(* CoDeSys 2.3.9.31 project: 1floor_2014_05_04.pr6 *)
(* Libraries: TcPlcUtilitiesBC.lb6 13.5.05 12:19:40, PlcSystemBC.lb6 21.3.01 12:03:02, TcAdsBC.lb6 5.7.02 12:03:02, standard.lb6 5.6.98 12:03:02 *)

(* Global variable list: main *)
VAR_GLOBAL


(*ADS*)

	ads_adr1: STRING:='10.0.5.61.1.1';
	ads_adr2: STRING:='10.0.5.62.1.1';
	ads_adr3: STRING:='10.0.5.63.1.1';

	write_ads: ADSWRITE;

	data2floor: ARRAY[0..3] OF BYTE;
	data2floor_prev :ARRAY[0..3] OF BYTE;
	data3floor: ARRAY[0..10] OF BYTE;
	data3floor_prev :ARRAY[0..10] OF BYTE;

	m_fancoil_vitalnya_low 	AT%MX300.0: BOOL;
	m_fancoil_vitalnya_med 	AT%MX300.1: BOOL;
	m_fancoil_vitalnya_high 	AT%MX300.2: BOOL;
	skvazhyna 		AT%MX300.3:BOOL;
	tepla_pidloga		AT%MX300.4:BOOL;
	T_out3			AT%MB303:BYTE;


	iHour			AT%MB304:BYTE;
	iMinute			AT%MB305:BYTE;
	lights			AT%MB306:DWORD;

	sw_tambur2_1	AT%MX200.0:BOOL;
	sw_tambur3_2	AT%MX300.1:BOOL;
	bDarkOutside		AT%MX300.6:BOOL;
	bT_out_sign		AT%MX300.7:BOOL;

	eib_komora_l 						AT%MX400.0:BOOL;
	eib_su1_l 							AT%MX400.1:BOOL;
	eib_topochna_l 						AT%MX400.2:BOOL;
	eib_su2_bra	 						AT%MX400.3:BOOL;
	eib_topochna2_l 						AT%MX400.4:BOOL;
	eib_su2_l 							AT%MX400.5:BOOL;
	eib_su1_rakovyna 					AT%MX400.6:BOOL;
	eib_su2_dush 						AT%MX400.7:BOOL;
	eib_dush 							AT%MX401.0:BOOL;
	eib_vitalnya_smugy2 					AT%MX401.1:BOOL;
	eib_su2_polytsi 						AT%MX401.2:BOOL;
	eib_kuhnya1	 						AT%MX401.3:BOOL;
	eib_kuhnya2	 						AT%MX401.4:BOOL;
	eib_vitalnya_smugy1 					AT%MX401.5:BOOL;
	eib_vitalnya_l 						AT%MX401.6:BOOL;
	eib_vitalnya_prokladka 				AT%MX401.7:BOOL;
	eib_terassa_stina	 					AT%MX402.0:BOOL;
	eib_pidval_shody	 					AT%MX402.1:BOOL;
	eib_terassa 							AT%MX402.2:BOOL;
	eib_skhody2pov 						AT%MX402.3:BOOL;
	eib_tambur_l 							AT%MX402.4:BOOL;

	eib_vent_su1 							AT%MX402.5:BOOL;
	eib_vent_kuh_low 						AT%MX402.6:BOOL;
	eib_vent_dush 						AT%MX402.7:BOOL;
	eib_vent_komora 						AT%MX403.0:BOOL;
	eib_vent_kuh_high 					AT%MX403.1:BOOL;

END_VAR

(* Global variable list: physical *)
VAR_GLOBAL
(*din1_1*)moove_su1		AT %IX80.0:	BOOL;
(*din1_2*)moove_topochna	AT %IX80.1:	BOOL;
(*din1_3*)moove_su2	AT %IX80.2:	BOOL;
(*din1_4*)moove_korydor_ops	AT %IX80.3:	BOOL;
(*din1_5*)moove_korydor	AT %IX80.4:	BOOL;
(*din1_6*)moove_vitalnya	AT %IX80.5:	BOOL;
(*din1_7*)moove_komora	AT %IX80.6:	BOOL;
	din1_8	AT %IX80.7:	BOOL;
(*din2_1*)moove_kino		AT %IX81.0:	BOOL;
(*din2_2*)moove_skhody2_3	AT %IX81.1:	BOOL;
(*din2_3*)moove_skhody1_2	AT %IX81.2:	BOOL;
(*din2_4*)moove_garderob	AT %IX81.3:	BOOL;
(*din2_5*)moove_studio		AT %IX81.4:	BOOL;
(*din2_6*)moove_tambur3	AT %IX81.5:	BOOL;
(*din2_7*)moove_kabinet	AT %IX81.6:	BOOL;
(*din2_8*)moove_dytjacha	AT %IX81.7:	BOOL;
(*din3_1*)moove_spalnya	AT %IX82.0:	BOOL;
	din3_2	AT %IX82.1:	BOOL;
(*din3_3*)moove_korydor3	AT %IX82.2:	BOOL;
	din3_4	AT %IX82.3:	BOOL;
	din3_5	AT %IX82.4:	BOOL;
	din3_6	AT %IX82.5:	BOOL;
	din3_7	AT %IX82.6:	BOOL;
	(*din3_8sw_vhid2		AT %IX82.7:	BOOL;*)
	din4_1	AT %IX83.0:	BOOL;
	(*din4_2*)sw_su1_2		AT %IX83.1:	BOOL;
	(*din4_3*)sw_komora1		AT %IX83.2:	BOOL;
	(*din4_4*)sw_vhid1		AT %IX83.3:	BOOL;
	(*din4_5*)sw_topochna2	AT %IX83.4:	BOOL;
	sw_vhid2					AT %IX83.5:	BOOL;
	(*din4_7*)sw_topochna1	AT %IX83.6:	BOOL;
	(*din4_8*)sw_su1_1		AT %IX83.7:	BOOL;
	(*din5_1*)sw_tambur1_2	AT %IX84.0:	BOOL;
	(*din5_2*)sw_su2			AT %IX84.1:	BOOL;
	(*din5_3*)sw_kuh_su2		AT %IX84.2:	BOOL;
	(*din5_4*)sw_kuh3			AT %IX84.3:	BOOL;
	din5_5					AT %IX84.4:	BOOL;
	(*din5_6*)sw_kuh4			AT %IX84.5:	BOOL;
	(*din5_7*)sw_tambur1		AT %IX84.6:	BOOL;
	(*din5_8*)sw_vitalnya1		AT %IX84.7:	BOOL;
	(*din6_1*)sw_vitalnya2		AT %IX85.0:	BOOL;
	(*din6_2*)sw_kuh2			AT %IX85.1:	BOOL;
	din6_3					AT %IX85.2:	BOOL;
	(*din6_4*)sw_kuh1			AT %IX85.3:	BOOL;
	(*din6_5*)sw_vitalnya3		AT %IX85.4:	BOOL;
	(*din6_6*)sw_tambur3		AT %IX85.5:	BOOL;
	(*din6_7*)sw_tambur_su	AT %IX85.6:	BOOL;
	(*din6_8*)sw_transit2pov	AT %IX85.7:	BOOL;

(*din7_1*)ch_sensor1	AT %IX86.0:	BOOL;
(*din7_2*)ch_sensor2	AT %IX86.1:	BOOL;
(*din7_3*)zatoplennya_kot	AT %IX86.2:	BOOL;
(*din7_4*)zatoplennya_komora	AT %IX86.3:	BOOL;
(*din7_5*)zatoplennya_su2	AT %IX86.4:	BOOL;
(*din7_6*)zatoplennya_kuh	AT %IX86.5:	BOOL;
(*din7_7*)zatoplennya_su3pov	AT %IX86.6:	BOOL;
	din7_8	AT %IX86.7:	BOOL;

	(*dout1_1*)komora_l			AT %QX80.0:	BOOL;
	(*dout1_2*)su1_l				AT %QX80.1:	BOOL;
	(*dout1_3*)topochna_l			AT %QX80.2:	BOOL;
	(*dout1_4*)su2_bra			AT %QX80.3:	BOOL;
	(*dout1_5*)topochna2_l			AT %QX80.4:	BOOL;
	(*dout1_6*)su2_l				AT %QX80.5:	BOOL;
	(*dout1_7*)su1_rakovyna		AT %QX80.6:	BOOL;
	(*dout1_8*)su2_dush			AT %QX80.7:	BOOL;
	(*dout2_1*)dush				AT %QX81.0:	BOOL;
	(*dout2_2*)vitalnya_smugy2		AT %QX81.1:	BOOL;
	(*dout2_3*) su2_polytsi			AT %QX81.2:	BOOL;
	(*dout2_4*)fancoil_vitalnya_low			AT %QX81.3:	BOOL;
	(*dout2_5*)kuhnya1			AT %QX81.4:	BOOL;
	(*dout2_6*)fancoil_vitalnya_med			AT %QX81.5:	BOOL;
	(*dout2_7*)kuhnya2			AT %QX81.6:	BOOL;
	(*dout2_8*)fancoil_vitalnya_high		AT %QX81.7:	BOOL;
	w_valve_recirc	AT %QX82.0:	BOOL;
	dout3_2	AT %QX82.1:	BOOL;
	w_valve3pov	AT %QX82.2:	BOOL;
	(*dout3_4*)vitalnya_smugy1		AT %QX82.3:	BOOL;
	w_valve1pov	AT %QX82.4:	BOOL;
	(*dout3_6*)vitalnya_l			AT %QX82.5:	BOOL;
	(*dout3_7*)freecooling	AT %QX82.6:	BOOL;
	(*dout3_8*)vitalnya_prokladka	AT %QX82.7:	BOOL;
	(*dout4_1*)terassa_stina		AT %QX83.0:	BOOL;
	(*dout4_2*)pidval_shody		AT %QX83.1:	BOOL;
	(*dout4_3*)terassa				AT %QX83.2:	BOOL;
	(*dout4_4*)skhody2pov			AT %QX83.3:	BOOL;
	dout4_5	AT %QX83.4:	BOOL;
	dout4_6	AT %QX83.5:	BOOL;
	dout4_7	AT %QX83.6:	BOOL;
	(*dout4_8*)tambur_l			AT %QX83.7:	BOOL;
	dout5_1	AT %QX84.0:	BOOL;
	dout5_2 AT %QX84.1:	BOOL;
(*dout5_3*)gas_valve	AT %QX84.2:	BOOL;
	dout5_4	AT %QX84.3:	BOOL;
	dout5_5	AT %QX84.4:	BOOL;
	dout5_6	AT %QX84.5:	BOOL;
	dout5_7	AT %QX84.6:	BOOL;
	dout5_8	AT %QX84.7:	BOOL;
	dout6_1	AT %QX85.0:	BOOL;
	dout6_2	AT %QX85.1:	BOOL;
	dout6_3	AT %QX85.2:	BOOL;
	dout6_4	AT %QX85.3:	BOOL;
	dout6_5	AT %QX85.4:	BOOL;
	dout6_6	AT %QX85.5:	BOOL;
	dout6_7	AT %QX85.6:	BOOL;
	dout6_8	AT %QX85.7:	BOOL;
	dout7_1	AT %QX86.0:	BOOL;
	dout7_2	AT %QX86.1:	BOOL;
	dout7_3	AT %QX86.2:	BOOL;
	dout7_4	AT %QX86.3:	BOOL;
	dout7_5	AT %QX86.4:	BOOL;
	dout7_6	AT %QX86.5:	BOOL;
	dout7_7	AT %QX86.6:	BOOL;
	dout7_8	AT %QX86.7:	BOOL;
	dout8_1	AT %QX87.0:	BOOL;
	dout8_2	AT %QX87.1:	BOOL;
	dout8_3	AT %QX87.2:	BOOL;
	dout8_4	AT %QX87.3:	BOOL;
	dout8_5	AT %QX87.4:	BOOL;
	dout8_6	AT %QX87.5:	BOOL;
	dout8_7	AT %QX87.6:	BOOL;
	dout8_8	AT %QX87.7:	BOOL;
	(*dout9_1*)vent_su1		AT %QX88.0:	BOOL;
	(*dout9_2*)vent_kuh_low	AT %QX88.1:	BOOL;
	(*dout9_3*)vent_dush		AT %QX88.2:	BOOL;
	(*dout9_4*)collector_komora		AT %QX88.3:	BOOL;
	(*dout9_5*)vent_komora	AT %QX88.4:	BOOL;
	(*dout9_6	*)collector_kuh		AT %QX88.5:	BOOL;
	(*dout9_7*)vent_kuh_high	AT %QX88.6:	BOOL;
	(*dout9_8*)collector_vitalnya1	AT %QX88.7:	BOOL;
	(*dout10_1*)collector_vitalnya2	AT %QX89.0:	BOOL;
	dout10_2	AT %QX89.1:	BOOL;
	(*dout10_3*)collector_su2		AT %QX89.2:	BOOL;
	dout10_4	AT %QX89.3:	BOOL;
	(*dout10_5*)collector_vhid_stina	AT %QX89.4:	BOOL;
	dout10_6	AT %QX89.5:	BOOL;
	(*dout10_7*)collector_vhid		AT %QX89.6:	BOOL;
	dout10_8	AT %QX89.7:	BOOL;
	dout11_1	AT %QX90.0:	BOOL;
	dout11_2	AT %QX90.1:	BOOL;
	dout11_3	AT %QX90.2:	BOOL;
	dout11_4	AT %QX90.3:	BOOL;
	dout11_5	AT %QX90.4:	BOOL;
	dout11_6	AT %QX90.5:	BOOL;
	dout11_7	AT %QX90.6:	BOOL;
	dout11_8	AT %QX90.7:	BOOL;

	klapan_vitalnya	AT %QB2:	INT;
	KL4414_2_Out	AT %QB6:	INT;
	KL4414_3_Out	AT %QB10:	INT;
	KL4414_4_Out	AT %QB14:	INT;

	temp_vhid	AT %IB50:	INT; (*25*)
	temp_dush	AT %IB58:	INT;(*25*)
	temp_kuh	AT %IB66:	INT;(*-136*)
	temp_vhid_stina	AT %IB70:	INT;(*0*)
(*
(* @GLOBAL_VARIABLE_LIST := TwinCAT_Import *)
(* @PATH := '' *)
VAR_GLOBAL (* DO NOT CHANGE THIS SHEET MANUALLY! *)
	PlcInVar_0	AT %QB128:	USINT;
	PlcInVar_1	AT %QB129:	USINT;
	PlcInVar_2	AT %QB130:	USINT;
	PlcInVar_3	AT %QB131:	USINT;
	PlcInVar_4	AT %QB132:	USINT;
	PlcInVar_5	AT %QB133:	USINT;
	PlcInVar_6	AT %QB134:	USINT;
	PlcInVar_7	AT %QB135:	USINT;
	PlcInVar_8	AT %QB136:	USINT;
	PlcInVar_9	AT %QB137:	USINT;
	PlcInVar_10	AT %QB138:	USINT;
	PlcInVar_11	AT %QB139:	USINT;
	PlcInVar_12	AT %QB140:	USINT;
	PlcInVar_13	AT %QB141:	USINT;
	PlcInVar_14	AT %QB142:	USINT;
	PlcInVar_15	AT %QB143:	USINT;
	PlcOutVar_0	AT %IB128:	USINT;
	PlcOutVar_1	AT %IB129:	USINT;
	PlcOutVar_2	AT %IB130:	USINT;
	PlcOutVar_3	AT %IB131:	USINT;
	PlcOutVar_4	AT %IB132:	USINT;
	PlcOutVar_5	AT %IB133:	USINT;
	PlcOutVar_6	AT %IB134:	USINT;
	PlcOutVar_7	AT %IB135:	USINT;
	PlcOutVar_8	AT %IB136:	USINT;
	PlcOutVar_9	AT %IB137:	USINT;
	PlcOutVar_10	AT %IB138:	USINT;
	PlcOutVar_11	AT %IB139:	USINT;
	PlcOutVar_12	AT %IB140:	USINT;
	PlcOutVar_13	AT %IB141:	USINT;
	PlcOutVar_14	AT %IB142:	USINT;
	PlcOutVar_15	AT %IB143:	USINT;
	Term_2_KL4414_1_State	AT %IB0:	USINT;
	Term_2_KL4414_1_Data_In	AT %IB2:	INT;
	Term_2_KL4414_1_Ctrl	AT %QB0:	USINT;
	Term_2_KL4414_1_Data_Out	AT %QB2:	INT;
	Term_2_KL4414_2_State	AT %IB4:	USINT;
	Term_2_KL4414_2_Data_In	AT %IB6:	INT;
	Term_2_KL4414_2_Ctrl	AT %QB4:	USINT;
	Term_2_KL4414_2_Data_Out	AT %QB6:	INT;
	Term_2_KL4414_3_State	AT %IB8:	USINT;
	Term_2_KL4414_3_Data_In	AT %IB10:	INT;
	Term_2_KL4414_3_Ctrl	AT %QB8:	USINT;
	Term_2_KL4414_3_Data_Out	AT %QB10:	INT;
	Term_2_KL4414_4_State	AT %IB12:	USINT;
	Term_2_KL4414_4_Data_In	AT %IB14:	INT;
	Term_2_KL4414_4_Ctrl	AT %QB12:	USINT;
	Term_2_KL4414_4_Data_Out	AT %QB14:	INT;
	Term_14_KL3228_4_1_State	AT %IB16:	USINT;
	Term_14_KL3228_4_1_Data_In	AT %IB18:	INT;
	Term_14_KL3228_4_1_Ctrl	AT %QB16:	USINT;
	Term_14_KL3228_4_1_Data_Out	AT %QB18:	INT;
	Term_14_KL3228_4_2_State	AT %IB20:	USINT;
	Term_14_KL3228_4_2_Data_In	AT %IB22:	INT;
	Term_14_KL3228_4_2_Ctrl	AT %QB20:	USINT;
	Term_14_KL3228_4_2_Data_Out	AT %QB22:	INT;
	Term_14_KL3228_4_3_State	AT %IB24:	USINT;
	Term_14_KL3228_4_3_Data_In	AT %IB26:	INT;
	Term_14_KL3228_4_3_Ctrl	AT %QB24:	USINT;
	Term_14_KL3228_4_3_Data_Out	AT %QB26:	INT;
	Term_14_KL3228_4_4_State	AT %IB28:	USINT;
	Term_14_KL3228_4_4_Data_In	AT %IB30:	INT;
	Term_14_KL3228_4_4_Ctrl	AT %QB28:	USINT;
	Term_14_KL3228_4_4_Data_Out	AT %QB30:	INT;
	Term_15_KL3228_4_1_State	AT %IB32:	USINT;
	Term_15_KL3228_4_1_Data_In	AT %IB34:	INT;
	Term_15_KL3228_4_1_Ctrl	AT %QB32:	USINT;
	Term_15_KL3228_4_1_Data_Out	AT %QB34:	INT;
	Term_15_KL3228_4_2_State	AT %IB36:	USINT;
	Term_15_KL3228_4_2_Data_In	AT %IB38:	INT;
	Term_15_KL3228_4_2_Ctrl	AT %QB36:	USINT;
	Term_15_KL3228_4_2_Data_Out	AT %QB38:	INT;
	Term_15_KL3228_4_3_State	AT %IB40:	USINT;
	Term_15_KL3228_4_3_Data_In	AT %IB42:	INT;
	Term_15_KL3228_4_3_Ctrl	AT %QB40:	USINT;
	Term_15_KL3228_4_3_Data_Out	AT %QB42:	INT;
	Term_15_KL3228_4_4_State	AT %IB44:	USINT;
	Term_15_KL3228_4_4_Data_In	AT %IB46:	INT;
	Term_15_KL3228_4_4_Ctrl	AT %QB44:	USINT;
	Term_15_KL3228_4_4_Data_Out	AT %QB46:	INT;
	Term_16_KL3228_4_1_State	AT %IB48:	USINT;
	Term_16_KL3228_4_1_Data_In	AT %IB50:	INT;
	Term_16_KL3228_4_1_Ctrl	AT %QB48:	USINT;
	Term_16_KL3228_4_1_Data_Out	AT %QB50:	INT;
	Term_16_KL3228_4_2_State	AT %IB52:	USINT;
	Term_16_KL3228_4_2_Data_In	AT %IB54:	INT;
	Term_16_KL3228_4_2_Ctrl	AT %QB52:	USINT;
	Term_16_KL3228_4_2_Data_Out	AT %QB54:	INT;
	Term_16_KL3228_4_3_State	AT %IB56:	USINT;
	Term_16_KL3228_4_3_Data_In	AT %IB58:	INT;
	Term_16_KL3228_4_3_Ctrl	AT %QB56:	USINT;
	Term_16_KL3228_4_3_Data_Out	AT %QB58:	INT;
	Term_16_KL3228_4_4_State	AT %IB60:	USINT;
	Term_16_KL3228_4_4_Data_In	AT %IB62:	INT;
	Term_16_KL3228_4_4_Ctrl	AT %QB60:	USINT;
	Term_16_KL3228_4_4_Data_Out	AT %QB62:	INT;
	Term_17_KL3228_4_1_State	AT %IB64:	USINT;
	Term_17_KL3228_4_1_Data_In	AT %IB66:	INT;
	Term_17_KL3228_4_1_Ctrl	AT %QB64:	USINT;
	Term_17_KL3228_4_1_Data_Out	AT %QB66:	INT;
	Term_17_KL3228_4_2_State	AT %IB68:	USINT;
	Term_17_KL3228_4_2_Data_In	AT %IB70:	INT;
	Term_17_KL3228_4_2_Ctrl	AT %QB68:	USINT;
	Term_17_KL3228_4_2_Data_Out	AT %QB70:	INT;
	Term_17_KL3228_4_3_State	AT %IB72:	USINT;
	Term_17_KL3228_4_3_Data_In	AT %IB74:	INT;
	Term_17_KL3228_4_3_Ctrl	AT %QB72:	USINT;
	Term_17_KL3228_4_3_Data_Out	AT %QB74:	INT;
	Term_17_KL3228_4_4_State	AT %IB76:	USINT;
	Term_17_KL3228_4_4_Data_In	AT %IB78:	INT;
	Term_17_KL3228_4_4_Ctrl	AT %QB76:	USINT;
	Term_17_KL3228_4_4_Data_Out	AT %QB78:	INT; 
	Term_3_KL2408_1_Output	AT %QX80.0:	BOOL;
	Term_3_KL2408_2_Output	AT %QX80.1:	BOOL;
	Term_3_KL2408_3_Output	AT %QX80.2:	BOOL;
	Term_3_KL2408_4_Output	AT %QX80.3:	BOOL;
	Term_3_KL2408_5_Output	AT %QX80.4:	BOOL;
	Term_3_KL2408_6_Output	AT %QX80.5:	BOOL;
	Term_3_KL2408_7_Output	AT %QX80.6:	BOOL;
	Term_3_KL2408_8_Output	AT %QX80.7:	BOOL;
	Term_4_KL2408_1_Output	AT %QX81.0:	BOOL;
	Term_4_KL2408_2_Output	AT %QX81.1:	BOOL;
	Term_4_KL2408_3_Output	AT %QX81.2:	BOOL;
	Term_4_KL2408_4_Output	AT %QX81.3:	BOOL;
	Term_4_KL2408_5_Output	AT %QX81.4:	BOOL;
	Term_4_KL2408_6_Output	AT %QX81.5:	BOOL;
	Term_4_KL2408_7_Output	AT %QX81.6:	BOOL;
	Term_4_KL2408_8_Output	AT %QX81.7:	BOOL;
	Term_5_KL2408_1_Output	AT %QX82.0:	BOOL;
	Term_5_KL2408_2_Output	AT %QX82.1:	BOOL;
	Term_5_KL2408_3_Output	AT %QX82.2:	BOOL;
	Term_5_KL2408_4_Output	AT %QX82.3:	BOOL;
	Term_5_KL2408_5_Output	AT %QX82.4:	BOOL;
	Term_5_KL2408_6_Output	AT %QX82.5:	BOOL;
	Term_5_KL2408_7_Output	AT %QX82.6:	BOOL;
	Term_5_KL2408_8_Output	AT %QX82.7:	BOOL;
	Term_6_KL2408_1_Output	AT %QX83.0:	BOOL;
	Term_6_KL2408_2_Output	AT %QX83.1:	BOOL;
	Term_6_KL2408_3_Output	AT %QX83.2:	BOOL;
	Term_6_KL2408_4_Output	AT %QX83.3:	BOOL;
	Term_6_KL2408_5_Output	AT %QX83.4:	BOOL;
	Term_6_KL2408_6_Output	AT %QX83.5:	BOOL;
	Term_6_KL2408_7_Output	AT %QX83.6:	BOOL;
	Term_6_KL2408_8_Output	AT %QX83.7:	BOOL;
	Term_7_KL2408_1_Output	AT %QX84.0:	BOOL;
	Term_7_KL2408_2_Output	AT %QX84.1:	BOOL;
	Term_7_KL2408_3_Output	AT %QX84.2:	BOOL;
	Term_7_KL2408_4_Output	AT %QX84.3:	BOOL;
	Term_7_KL2408_5_Output	AT %QX84.4:	BOOL;
	Term_7_KL2408_6_Output	AT %QX84.5:	BOOL;
	Term_7_KL2408_7_Output	AT %QX84.6:	BOOL;
	Term_7_KL2408_8_Output	AT %QX84.7:	BOOL;
	Term_8_KL2408_1_Output	AT %QX85.0:	BOOL;
	Term_8_KL2408_2_Output	AT %QX85.1:	BOOL;
	Term_8_KL2408_3_Output	AT %QX85.2:	BOOL;
	Term_8_KL2408_4_Output	AT %QX85.3:	BOOL;
	Term_8_KL2408_5_Output	AT %QX85.4:	BOOL;
	Term_8_KL2408_6_Output	AT %QX85.5:	BOOL;
	Term_8_KL2408_7_Output	AT %QX85.6:	BOOL;
	Term_8_KL2408_8_Output	AT %QX85.7:	BOOL;
	Term_9_KL2408_1_Output	AT %QX86.0:	BOOL;
	Term_9_KL2408_2_Output	AT %QX86.1:	BOOL;
	Term_9_KL2408_3_Output	AT %QX86.2:	BOOL;
	Term_9_KL2408_4_Output	AT %QX86.3:	BOOL;
	Term_9_KL2408_5_Output	AT %QX86.4:	BOOL;
	Term_9_KL2408_6_Output	AT %QX86.5:	BOOL;
	Term_9_KL2408_7_Output	AT %QX86.6:	BOOL;
	Term_9_KL2408_8_Output	AT %QX86.7:	BOOL;
	Term_10_KL2408_1_Output	AT %QX87.0:	BOOL;
	Term_10_KL2408_2_Output	AT %QX87.1:	BOOL;
	Term_10_KL2408_3_Output	AT %QX87.2:	BOOL;
	Term_10_KL2408_4_Output	AT %QX87.3:	BOOL;
	Term_10_KL2408_5_Output	AT %QX87.4:	BOOL;
	Term_10_KL2408_6_Output	AT %QX87.5:	BOOL;
	Term_10_KL2408_7_Output	AT %QX87.6:	BOOL;
	Term_10_KL2408_8_Output	AT %QX87.7:	BOOL;
	Term_11_KL2408_1_Output	AT %QX88.0:	BOOL;
	Term_11_KL2408_2_Output	AT %QX88.1:	BOOL;
	Term_11_KL2408_3_Output	AT %QX88.2:	BOOL;
	Term_11_KL2408_4_Output	AT %QX88.3:	BOOL;
	Term_11_KL2408_5_Output	AT %QX88.4:	BOOL;
	Term_11_KL2408_6_Output	AT %QX88.5:	BOOL;
	Term_11_KL2408_7_Output	AT %QX88.6:	BOOL;
	Term_11_KL2408_8_Output	AT %QX88.7:	BOOL;
	Term_12_KL2408_1_Output	AT %QX89.0:	BOOL;
	Term_12_KL2408_2_Output	AT %QX89.1:	BOOL;
	Term_12_KL2408_3_Output	AT %QX89.2:	BOOL;
	Term_12_KL2408_4_Output	AT %QX89.3:	BOOL;
	Term_12_KL2408_5_Output	AT %QX89.4:	BOOL;
	Term_12_KL2408_6_Output	AT %QX89.5:	BOOL;
	Term_12_KL2408_7_Output	AT %QX89.6:	BOOL;
	Term_12_KL2408_8_Output	AT %QX89.7:	BOOL;
	Term_13_KL2408_1_Output	AT %QX90.0:	BOOL;
	Term_13_KL2408_2_Output	AT %QX90.1:	BOOL;
	Term_13_KL2408_3_Output	AT %QX90.2:	BOOL;
	Term_13_KL2408_4_Output	AT %QX90.3:	BOOL;
	Term_13_KL2408_5_Output	AT %QX90.4:	BOOL;
	Term_13_KL2408_6_Output	AT %QX90.5:	BOOL;
	Term_13_KL2408_7_Output	AT %QX90.6:	BOOL;
	Term_13_KL2408_8_Output	AT %QX90.7:	BOOL;
	
END_VAR

*)
END_VAR

(* Data type *)
TYPE ROOM_HVAC :
STRUCT

	heat_mode:STRING;
	heat_speed:USINT;

	delta_t:SINT;
	t_cur:SINT;
	t_ust:SINT;

	fancoil_speed:SINT;
	klapan:WORD;

	collector1: BOOL;
	collector2: BOOL;
	collector3: BOOL;
	collector4: BOOL;

END_STRUCT
END_TYPE

(* POU MAIN, ST *)
PROGRAM MAIN
VAR

	i:INT;
END_VAR
zatoplennya;
light;
heat;
ADS_write;
END_PROGRAM

(* POU zatoplennya, ST *)
PROGRAM zatoplennya
VAR
END_VAR
w_valve1pov:=  (zatoplennya_komora OR zatoplennya_kuh OR zatoplennya_su2);
w_valve3pov:= (zatoplennya_su3pov);
w_valve_recirc:=zatoplennya_su3pov;
(*дописати код для перекривання води по сенсору в котельні та підвалі*)
(*СЕНСОР В КОТЕЛЬНЫЙ ВЫДКЛЮЧЕНИЙ ЧЕРЕЗ ПОСТЫЙНУ ВОЛОГЫСТЬ*)
gas_valve:=NOT (ch_sensor1 AND ch_sensor2);
END_PROGRAM

(* POU lights/light, ST *)
PROGRAM light
VAR
	komora1,topochna1, su1_1,su1_2, su2, tambur1,tambur2,tambur3, vhid1, vhid2, kuh1,kuh2,kuh3,kuh4,kuh_su2, vitalnya1,vitalnya2,vitalnya3:SWITCH;
	delay1, delay2: TIME;

	DUSH_M, SU1_M, KOMORA_M, TOPOCHNA_M:F_TRIG; (*задній фронт давачів руху*)
	su2_timer, su1_timer, topochna_timer, komora_timer:TOF;

	light_delay: TIME;
	su2_timer_started, su1_timer_started: BOOL;
	topochna_timer_started, komora_timer_started:BOOL;
	ZEBRA_TIMER:TOF;
	ZEBRA_SEMA:SEMA;
	ZEBRA_F: F_TRIG;

	DUSH2_TIMER: TOF;
	DUSH2_SEMA: SEMA;
	DUSH2_F: F_TRIG;
	fbDarkEdge:R_TRIG;

	prev_eib_komora_l 						:BOOL;
	prev_eib_su1_l 							:BOOL;
	prev_eib_topochna_l 						:BOOL;
	prev_eib_su2_bra	 						:BOOL;
	prev_eib_topochna2_l 						:BOOL;
	prev_eib_su2_l 							:BOOL;
	prev_eib_su1_rakovyna 					:BOOL;
	prev_eib_su2_dush 						:BOOL;
	prev_eib_dush 							:BOOL;
	prev_eib_vitalnya_smugy2 					:BOOL;
	prev_eib_su2_polytsi 						:BOOL;
	prev_eib_kuhnya1	 						:BOOL;
	prev_eib_kuhnya2	 						:BOOL;
	prev_eib_vitalnya_smugy1 					:BOOL;
	prev_eib_vitalnya_l 						:BOOL;
	prev_eib_vitalnya_prokladka 				:BOOL;
	prev_eib_terassa_stina	 				:BOOL;
	prev_eib_pidval_shody	 				:BOOL;
	prev_eib_terassa 							:BOOL;
	prev_eib_skhody2pov 						:BOOL;
	prev_eib_tambur_l 						:BOOL;
	prev_eib_vent_su1 						:BOOL;
	prev_eib_vent_kuh_low 					:BOOL;
	prev_eib_vent_dush 						:BOOL;
	prev_eib_vent_komora 					:BOOL;
	prev_eib_vent_kuh_high 					:BOOL;


END_VAR
delay1:=t#500ms; (*скільки тримати кнопку для довгого натискання*)
delay2:=t#5m; (*затримка вимкнення вентиляторів в туалетах*)
light_delay:=t#3m; (*час роботи світильників, увімкнених по давачу руху*)


komora1(MODE:='light&vent', IN:=sw_komora1 XOR sw_topochna2, SWITCH_DELAY:=delay1, SHORT_OFF_DELAY:=delay2, LONG_OFF_DELAY:=delay2);
IF komora1.long THEN  vent_komora:=NOT  vent_komora ; END_IF;

topochna1(MODE:='light',SWITCH_DELAY:=delay1, IN:=sw_topochna1);

su1_1(MODE:='light&vent', IN:=sw_su1_1 XOR sw_tambur_su, SWITCH_DELAY:=delay1,SHORT_OFF_DELAY:=delay2, LONG_OFF_DELAY:=delay2);
su1_2(MODE:='light',SWITCH_DELAY:=delay1, IN:=sw_su1_2);
su2(MODE:='light&vent', IN:=sw_su2,SWITCH_DELAY:=delay1, SHORT_OFF_DELAY:=delay2, LONG_OFF_DELAY:=delay2);


IF prev_eib_tambur_l = eib_tambur_l THEN
	tambur1(MODE:='light',SWITCH_DELAY:=delay1, IN:=sw_tambur1 XOR sw_vhid1);
	ZEBRA_TIMER(IN:=NOT moove_korydor_ops, PT:=light_delay);
	ZEBRA_F(clk:=ZEBRA_TIMER.Q);
	ZEBRA_SEMA(CLAIM:=(NOT tambur_l AND tambur1.short ) OR (NOT moove_korydor_ops AND bDarkOutside), RELEASE:=(tambur_l AND tambur1.short) OR ZEBRA_f.Q);
	tambur_l:=ZEBRA_SEMA.BUSY;
ELSE
	tambur_l:=eib_tambur_l;
END_IF

(*skhody1:=tambur2.Q_LONG; (*для вимкнення світла на обох прольотах*) *)

tambur3(MODE:='light', SWITCH_DELAY:=delay1,IN:=sw_tambur3);

vhid2(MODE:='light', IN:=sw_vhid2);

kuh1(MODE:='light&vent', IN:=sw_kuh1,SWITCH_DELAY:=delay1, SHORT_OFF_DELAY:=delay2, LONG_OFF_DELAY:=delay2 );
kuh2(MODE:='light', SWITCH_DELAY:=delay1,IN:=sw_kuh2 XOR sw_vitalnya1);
kuh3(MODE:='light', SWITCH_DELAY:=delay1,IN:=sw_kuh3 XOR sw_vitalnya1);
kuh4(MODE:='light',SWITCH_DELAY:=delay1, IN:=sw_kuh4 XOR sw_vitalnya2);


vitalnya1(MODE:='light',SWITCH_DELAY:=delay1, IN:=sw_vitalnya1);
vitalnya2(MODE:='light', SWITCH_DELAY:=delay1,IN:=sw_vitalnya2);
vitalnya3(MODE:='light', SWITCH_DELAY:=delay1,IN:=sw_vitalnya3);


(*комора*)
IF eib_komora_l = prev_eib_komora_l THEN

	IF komora1.short THEN komora_l := NOT komora_l; END_IF;
	KOMORA_M(CLK:=moove_komora);

	IF KOMORA_M.Q AND NOT komora_l THEN (*спрацювання давача руху*)
		komora_timer_started:=1; (*прапор спрацювання таймера*)
	END_IF

	komora_timer(PT:=light_delay, IN:=KOMORA_M.Q);

	IF komora_timer_started  THEN (*якщо працює таймер, то тримати світло увімкненим*)
		IF komora1.Q_S_fall.Q  THEN
			komora_l:=FALSE;
			komora_timer_started:=FALSE;
		ELSE
			IF NOT komora_timer.Q THEN
				komora_timer_started:=FALSE;
			END_IF
			komora_l:=komora_timer.Q;
		END_IF
	END_IF
ELSE
	komora_l:=eib_komora_l;
END_IF

(*топочна*)

IF (eib_topochna_l= prev_eib_topochna_l) THEN

	TOPOCHNA_M(CLK:=moove_topochna);

	IF TOPOCHNA_M.Q AND NOT topochna2_l THEN (*спрацювання давача руху*)
		topochna_timer_started:=1; (*прапор спрацювання таймера*)
	END_IF

	topochna_timer(PT:=light_delay, IN:=TOPOCHNA_M.Q);

	IF topochna_timer_started  THEN (*якщо працює таймер, то тримати світло увімкненим*)
		IF topochna1.Q_S_fall.Q  THEN
			topochna_l:=FALSE;
			topochna_timer_started:=FALSE;
		ELSE
			IF NOT topochna_timer.Q THEN
				topochna_timer_started:=FALSE;
			END_IF
			topochna_l:=topochna_timer.Q;
		END_IF
	END_IF

	IF topochna1.short THEN
		topochna_l:=NOT topochna_l;
	END_IF;
ELSE
	topochna_l:= eib_topochna_l;
END_IF
topochna2_l:=topochna_l;


(*санвузол1*)


SU1_M(CLK:=moove_su1);
(*
	IF SU1_M.Q AND NOT su1_l THEN (*спрацювання давача руху*)
		su1_timer_started:=1; (*прапор спрацювання таймера*)
	END_IF

	su1_timer(PT:=light_delay, IN:=SU1_M.Q);

	IF su1_timer_started  THEN (*якщо працює таймер, то тримати світло увімкненим*)
		IF su1_1.Q_S_fall.Q THEN
			su1_l:=FALSE;
			su1_timer_started:=FALSE;
		ELSE
			IF NOT su1_timer.Q THEN
				su1_timer_started:=FALSE;
			END_IF
			su1_l:=su1_timer.Q;
		END_IF
	END_IF
*)
IF eib_su1_l=prev_eib_su1_l THEN
	IF su1_1.short THEN  su1_l:=NOT su1_l; END_IF;
ELSE
	su1_l:=eib_su1_l;
END_IF
IF eib_su1_rakovyna =prev_eib_su1_rakovyna THEN
	IF su1_2.short THEN su1_rakovyna:=NOT su1_rakovyna; END_IF;
ELSE
	eib_su1_rakovyna:=eib_su1_rakovyna;
END_IF

IF su1_1.long THEN vent_su1:=NOT vent_su1;END_IF;

IF (eib_su2_polytsi = prev_eib_su2_polytsi) OR (eib_dush=prev_eib_dush) THEN
	IF su2.short THEN
		IF NOT (su2_polytsi OR dush) THEN
			 su2_polytsi:=TRUE; dush:=TRUE;
		ELSE
			su2_polytsi:=FALSE; dush:=FALSE;
		END_IF
	END_IF
END_IF

IF eib_su2_polytsi <> prev_eib_su2_polytsi THEN su2_polytsi:=eib_su2_polytsi; END_IF
IF eib_dush<>prev_eib_dush THEN dush:=eib_dush; END_IF


IF su2.long THEN
vent_dush:=NOT vent_dush;
END_IF

(*tambur_l:=tambur1.Q_SHORT; *)
IF eib_pidval_shody= prev_eib_pidval_shody THEN
	pidval_shody:=tambur3.Q_SHORT;
ELSE
	pidval_shody:=eib_pidval_shody;
END_IF

IF eib_kuhnya1 = prev_eib_kuhnya1 THEN
	kuhnya1:=kuh1.Q_SHORT;
ELSE
	kuhnya1:=eib_kuhnya1;
END_IF

IF eib_kuhnya2 = prev_eib_kuhnya2 THEN
	kuhnya2:=kuh1.Q_SHORT;
ELSE
	kuhnya2:=eib_kuhnya2;
END_IF

vent_kuh_high:=kuh1.Q_LONG;

IF eib_vitalnya_smugy1= prev_eib_vitalnya_smugy1 THEN
	vitalnya_smugy1:=kuh2.Q_SHORT ;
ELSE
	vitalnya_smugy1:=eib_vitalnya_smugy1;
END_IF
IF eib_vitalnya_smugy2= prev_eib_vitalnya_smugy2 THEN
	vitalnya_smugy2:=kuh2.Q_SHORT ;
ELSE
	vitalnya_smugy2:=eib_vitalnya_smugy2;
END_IF

IF eib_vitalnya_prokladka = prev_eib_vitalnya_prokladka THEN
	vitalnya_prokladka:=kuh3.Q_SHORT;
ELSE
	vitalnya_prokladka:=eib_vitalnya_prokladka;
END_IF

dout4_7:=vitalnya_prokladka;

IF eib_vitalnya_l = prev_eib_vitalnya_l THEN
	vitalnya_l:=kuh4.Q_SHORT;
ELSE
	vitalnya_l:=eib_vitalnya_l;
END_IF

(*санвузол2 з душем*)
kuh_su2(MODE:='light&vent', IN:=sw_kuh_su2,SWITCH_DELAY:=delay1, SHORT_OFF_DELAY:=delay2, LONG_OFF_DELAY:=delay2);
(*DUSH2_TIMER(IN:=NOT moove_su2, PT:=light_delay);
DUSH2_F(clk:=DUSH2_TIMER.Q);
DUSH2_SEMA(CLAIM:=(NOT su2_l AND kuh_su2.short ) OR NOT moove_su2 , RELEASE:=(su2_l AND kuh_su2.short) OR DUSH2_f.Q);

su2_l:=DUSH2_SEMA.BUSY;
su2_dush:=DUSH2_SEMA.BUSY;
*)

IF (eib_su2_l=prev_eib_su2_l) OR (eib_su2_bra=prev_eib_su2_bra) THEN
	IF kuh_su2.short THEN
		IF NOT (su2_l OR su2_bra) THEN su2_l:=TRUE; su2_bra:=TRUE;
		ELSE su2_l:=FALSE; su2_bra:=FALSE;
		END_IF
	END_IF
END_IF

IF (eib_su2_l<>prev_eib_su2_l) THEN su2_l:=eib_su2_l; END_IF
IF (eib_su2_bra<>prev_eib_su2_bra) THEN su2_bra:=eib_su2_bra; END_IF

IF eib_su2_dush = prev_eib_su2_dush THEN
	IF kuh_su2.long THEN su2_dush:= NOT su2_dush;END_IF
ELSE
	su2_dush:=eib_su2_dush;
END_IF

IF (eib_terassa_stina=prev_eib_terassa_stina) OR (eib_terassa=prev_eib_terassa) THEN
	IF vitalnya3.short THEN
		terassa_stina:= NOT terassa_stina;
		terassa:=NOT terassa;
	END_IF
END_IF
IF (eib_terassa_stina=prev_eib_terassa_stina) THEN terassa_stina:=eib_terassa_stina;END_IF
IF (eib_terassa=prev_eib_terassa) THEN terassa:=eib_terassa;END_IF

(*сходи на 2й поверх*)
fbDarkEdge(CLK:=bDarkOutside);
IF eib_skhody2pov=prev_eib_skhody2pov THEN
	tambur2(MODE:='light',SWITCH_DELAY:=delay1, IN:=sw_tambur1_2 OR sw_tambur2_1);
	IF tambur2.short THEN  skhody2pov:=NOT skhody2pov; END_IF
ELSE
	skhody2pov:=eib_skhody2pov;
END_IF


	prev_eib_komora_l 						:=eib_komora_l ;
	prev_eib_su1_l 							:=eib_su1_l ;
	prev_eib_topochna_l 						:=eib_topochna_l ;
	prev_eib_su2_bra	 						:=eib_su2_bra;
	prev_eib_topochna2_l 						:=eib_topochna2_l;
	prev_eib_su2_l 							:=eib_su2_l ;
	prev_eib_su1_rakovyna 					:=eib_su1_rakovyna;
	prev_eib_su2_dush 						:=eib_su2_dush;
	prev_eib_dush 							:=eib_dush ;
	prev_eib_vitalnya_smugy2 					:=eib_vitalnya_smugy2 ;
	prev_eib_su2_polytsi 						:=eib_su2_polytsi ;
	prev_eib_kuhnya1	 						:=eib_kuhnya1;
	prev_eib_kuhnya2	 						:=eib_kuhnya2;
	prev_eib_vitalnya_smugy1 					:=eib_vitalnya_smugy1;
	prev_eib_vitalnya_l 						:=eib_vitalnya_l;
	prev_eib_vitalnya_prokladka 				:=eib_vitalnya_prokladka;
	prev_eib_terassa_stina	 				:=eib_terassa_stina;
	prev_eib_pidval_shody	 				:=eib_pidval_shody;
	prev_eib_terassa 							:=eib_terassa ;
	prev_eib_skhody2pov 						:=eib_skhody2pov;
	prev_eib_tambur_l 						:=eib_tambur_l;
	prev_eib_vent_su1 						:=eib_vent_su1;
	prev_eib_vent_kuh_low 					:=eib_vent_kuh_low;
	prev_eib_vent_dush 						:=eib_vent_dush ;
	prev_eib_vent_komora 					:=eib_vent_komora ;
	prev_eib_vent_kuh_high 					:=eib_vent_kuh_high ;





data2floor[0].0:=sw_tambur1_2;
data2floor[0].1:=sw_vhid2;

data2floor[1].0:=moove_kino;
data2floor[1].1:=moove_skhody1_2;
data2floor[1].2:=moove_studio;
data2floor[1].3:=moove_kabinet;


data3floor[0].0:=moove_garderob;
data3floor[0].1:=moove_tambur3;
data3floor[0].2:=moove_dytjacha;
data3floor[0].3:=moove_spalnya;
data3floor[0].4:=moove_korydor3;
data3floor[0].5:=moove_skhody2_3;

data3floor[1].0:=komora_l;
data3floor[1].1:=su1_l;
data3floor[1].2:=topochna_l;
data3floor[1].3:=su2_bra	;
data3floor[1].4:=topochna2_l;
data3floor[1].5:=su2_l;
data3floor[1].6:=su1_rakovyna;
data3floor[1].7:=su2_dush;
data3floor[2].0:=dush;
data3floor[2].1:=vitalnya_smugy2;
data3floor[2].2:=su2_polytsi;
data3floor[2].3:=kuhnya1	;
data3floor[2].4:=kuhnya2	;
data3floor[2].5:=vitalnya_smugy1;
data3floor[2].6:=vitalnya_l;
data3floor[2].7:=vitalnya_prokladka;
data3floor[3].0:=terassa_stina	;
data3floor[3].1:=pidval_shody	;
data3floor[3].2:=terassa;
data3floor[3].3:=skhody2pov;
data3floor[3].4:=tambur_l;
data3floor[3].5:=vent_su1;
data3floor[3].6:=vent_kuh_low;
data3floor[3].7:=vent_dush;
data3floor[4].0:=vent_komora;
data3floor[4].1:=vent_kuh_high;
END_PROGRAM

(* POU lights/SWITCH, ST *)
FUNCTION_BLOCK SWITCH
VAR_INPUT
	IN:BOOL;
	SWITCH_DELAY:TIME; (*різниця між коротким і довгим натисненням*)
	SHORT_OFF_DELAY, LONG_OFF_DELAY: TIME; (*час затримки вимкнення по короткому та довгому натисненню*)
	MODE:STRING; (*delayed, light, light&vent, short&long, delayed_short&long, *)
	NUMBER_OF_OUTS:INT;
END_VAR
VAR_OUTPUT
	Q_SHORT:BOOL:=FALSE;
	Q_SHORT_D: BOOL;(*вихід для вимкнення із затримкою, вмикається разом із виходом короткого натискання*)
	Q_LONG:BOOL:=FALSE;
	Q_LONG_D:BOOL; (*вихід для вимкнення із затримкою, вмикається разом із виходом довгого натискання*)
END_VAR
VAR
	STAN:BOOL:=FALSE;
	Q_S_fall:F_TRIG; (*ловить задній фронт вихода короткого натискання*)
	Q_S_rise:F_TRIG; (*ловить задній фронт вихода короткого натискання*)
	Q_L_fall:F_TRIG;(*ловить задній фронт вихода довгого натискання*)
	chas: TIME; (*час доки кнопка натиснена*)

	long: BOOL; (*стає тру, якщо було довге натиснення*)
	short: BOOL; (*стає тру, якщо було коротке натиснення*)
	timer, short_off_delay_timer, long_off_delay_timer: TON; (*таймери: час натискання, час переключення відкладеного виходу по довгому та короткому натисканнях*)
	up: BOOL; (*кнопка натиснена*)

	delay_l, delay_s:BOOL; (*запускати таймери відкладеного вимкнення*)

	turn_off_long: BOOL;
	start_l, start_s:BOOL;
END_VAR
short:=0;
long:=0;
timer(IN:=IN AND STAN, PT:=t#10s);
IF IN AND STAN THEN
	chas:=timer.ET;
	up:=1;
ELSE
up:=0;
END_IF;

IF NOT IN AND NOT STAN THEN
chas:=t#0ms;
END_IF;

IF STAN AND NOT IN THEN
	IF chas <SWITCH_DELAY THEN
		short:=1;
		Q_SHORT:= NOT Q_SHORT;
	END_IF;
	IF chas>=SWITCH_DELAY THEN
		Q_LONG:= NOT Q_LONG;
		long:=1;
	END_IF;
END_IF;

(*затримка вимикання*)
Q_L_fall(CLK:=Q_LONG);
Q_S_fall(CLK:=Q_SHORT);
Q_S_rise(CLK:=Q_SHORT);

IF Q_L_FALL.Q THEN
		start_l:=TRUE;
END_IF

IF Q_S_FALL.Q THEN
	start_s:=TRUE;
END_IF

IF MODE='light&vent' THEN
	IF start_s THEN start_l:=start_s; END_IF
END_IF

IF LONG_OFF_DELAY <> t#0ms THEN (*виконувати лише якщо в блок переданий параметр затримки на вимкнення*)

	IF Q_LONG THEN
		Q_LONG_D:=Q_LONG;
	END_IF

	long_off_delay_timer(IN:=start_l, PT:=LONG_OFF_DELAY);

	IF long_off_delay_timer.Q THEN
		Q_LONG_D:=FALSE;
		start_l:=FALSE;
	END_IF

ELSE
	Q_LONG_D:=Q_LONG;
END_IF

IF SHORT_OFF_DELAY <> t#0ms THEN (*виконувати лише якщо в блок переданий параметр затримки на вимкнення*)

	IF Q_SHORT THEN
		Q_SHORT_D:=Q_SHORT;
	END_IF

	short_off_delay_timer(IN:=start_s, PT:=SHORT_OFF_DELAY);

	IF short_off_delay_timer.Q THEN
		Q_SHORT_D:=FALSE;
		start_s:=FALSE;
	END_IF


ELSE
	Q_SHORT_D:=Q_SHORT;
END_IF

IF MODE='delayed' THEN
	Q_LONG:=Q_LONG_D;
	Q_SHORT:=Q_SHORT_D;
END_IF
(*працють лише короткі замикання*)
IF MODE='light' THEN
	Q_SHORT_D:=FALSE;
	Q_LONG:=Q_SHORT;
	Q_LONG_D:=FALSE;
END_IF
(*затримки не працюють*)
IF MODE='short&long' THEN
	Q_SHORT_D:=FALSE;
	Q_LONG_D:=FALSE;
END_IF
(*при вимкненні всього світла вимикати вентилятор і затримкою*)
IF MODE='light&vent' THEN
	IF NOT Q_SHORT AND Q_LONG THEN
		Q_LONG:=Q_LONG_D;
	END_IF
END_IF

STAN := IN;
END_FUNCTION_BLOCK

(* POU heat, ST *)
PROGRAM heat
VAR
	temp_measure: TOF;
	t_vhid: REAL;
	t_dush: REAL;
	t_kuh: REAL;
	t_vhid_stina: REAL;

	t_max: SINT;
	t_min: SINT;
	t_out: REAL;
	i: INT;
	t_vhid_sum: REAL;
	t_dush_sum: REAL;
	t_vhid_stina_sum: REAL;
	t_kuh_sum: REAL;

	t_vhidPrev: REAL;
	t_dushPrev: REAL;
	t_vhid_stinaPrev: REAL;
	t_kuhPrev: REAL;

	delta_kuh: REAL;
	delta_vhid_stina: REAL;
	delta_dush: REAL;
	delta_vhid: REAL;
	retry:BOOL:=TRUE;(*переміряти температуру*)
	iRetryCounter: INT;
END_VAR
t_min:=0;
IF bT_out_sign THEN t_out:=0-t_out3; ELSE t_out:=t_out3; END_IF;

IF t_out >=17 AND skvazhyna THEN
	freecooling:=TRUE; (*freecooling means cold water in the system. There's hot water if it's FALSE*)
ELSE
	freecooling:=FALSE;
END_IF

	fancoil_vitalnya_low:=m_fancoil_vitalnya_low;
	fancoil_vitalnya_med:=m_fancoil_vitalnya_med;
	fancoil_vitalnya_high:=m_fancoil_vitalnya_high;
(*клапан управляється з 3го поверху*)


(*фільтр показань сенсорів температури*)
CASE i OF
0..500: init;
ELSE
	IF retry THEN
		temp_measure.PT:=t#2s;
	ELSE
		temp_measure.PT:=t#5m;
	END_IF
	IF retry THEN
		IF iRetryCounter >5 THEN iRetryCounter:=0; i:=0; ELSE iRetryCounter:=iRetryCounter+1; END_IF;
	END_IF;
	temp_measure( IN:=NOT temp_measure.q); (*перевіряти температуру кожні 20 хв*)

IF NOT temp_measure.Q THEN

	delta_kuh:=ABS(t_kuhPrev-temp_kuh*0.1);
	delta_vhid_stina:=ABS(t_vhid_stinaPrev-temp_vhid_stina*0.1);
	delta_dush:=ABS(t_dushPrev-temp_dush*0.1);
	delta_vhid:=ABS(t_vhidPrev-temp_vhid*0.1);
	retry:=FALSE;
	IF delta_kuh<1 THEN
		t_kuh:= temp_kuh * 0.1;
	ELSE
		t_kuh:=t_kuhPrev;
		retry:=TRUE;
	END_IF

	IF delta_vhid_stina<1 THEN
		t_vhid_stina:= temp_vhid_stina * 0.1;
	ELSE
		t_vhid_stina:=t_vhid_stinaPrev;
		retry:=TRUE;
	END_IF

	IF delta_dush<1 THEN
		t_dush:= temp_dush * 0.1;
	ELSE
		t_dush:=t_dushPrev;
		retry:=TRUE;
	END_IF

	IF delta_vhid<1 THEN
		t_vhid:= temp_vhid * 0.1;
	ELSE
		t_vhid:=t_vhidPrev;
		retry:=TRUE;
	END_IF

	t_kuhPrev:=t_kuh;
	t_vhid_stinaPrev:=t_vhid_stina;
	t_dushPrev:=t_dush;
	t_vhidPrev:=t_vhid;

END_IF
END_CASE

IF t_out>12 THEN
	t_max:=t_min;
ELSE
	IF t_out >0 THEN
		t_max:=10;
	ELSE
		t_max:=35;
	END_IF
END_IF

	IF t_vhid >=t_max THEN
		collector_vhid:=0;
	END_IF

	IF t_vhid <t_min THEN
		collector_vhid:=1;
	END_IF

	IF t_vhid_stina >=t_max THEN
		collector_vhid_stina:=0;
	END_IF

	IF t_vhid_stina <t_min THEN
		collector_vhid_stina:=1;
	END_IF

	IF t_dush >=t_max THEN
		collector_su2:=0;
	END_IF

	IF t_dush <t_min THEN
		collector_su2:=1;
	END_IF

	IF t_kuh<t_min THEN (*відкрити колектори, якщо підлога холодніша нижньої межі*)
		collector_vitalnya1:=1;
		collector_kuh:=1;
		collector_vitalnya2:=1;
	ELSE
		IF t_kuh >=t_max THEN (*закрити колектори, якщо підлога тепліша верхньої межі*)
			collector_vitalnya1:=0;
			collector_kuh:=0;
			collector_vitalnya2:=0;
			ELSE
				collector_vitalnya1:=tepla_pidloga;
				collector_kuh:=tepla_pidloga;
				collector_vitalnya2:=tepla_pidloga;
		END_IF
	END_IF
END_PROGRAM
ACTION init:
IF i=500 THEN
	t_vhidPrev:=t_vhid_sum/i;
	t_dushPrev:=t_dush_sum/i;
	t_vhid_stinaPrev:=t_vhid_stina_sum/i;
	t_kuhPrev:=t_kuh_sum/i;
	t_vhid_sum:=0;
	t_dush_sum:=0;
	t_vhid_stina_sum:=0;
	t_kuh_sum:=0;
	i:=501;
ELSE
	t_vhid_sum:=t_vhid_sum+temp_vhid*0.1;
	t_dush_sum:=t_dush_sum+temp_dush*0.1;
	t_vhid_stina_sum:=t_vhid_stina_sum+temp_vhid_stina*0.1;
	t_kuh_sum:=t_kuh_sum+temp_kuh*0.1;
	i:=i+1;
END_IF
END_ACTION

(* POU ADS_write, ST *)
PROGRAM ADS_write
VAR
	write_timeout: TIME;
	b_write3, b_write2: BOOL;
	write_ads3, write_ads2: ADSWRITE;

	timer3, timer2:TP;
	errorcounter3, errorcounter2, pack_c:CTU ;
	test_word: WORD;
	i,j,i1,j1: INT;
	data_changed: BOOL;
	try_again2, try_again3: BOOL;
	temp: INT;
	SENT2, SENT3:F_TRIG;
	SNT_CNT2, SNT_CNT3:CTU;
	fb_heartbeat_timer: TON;
END_VAR
write_timeout:=t#1s;
fb_heartbeat_timer(in:=NOT fb_heartbeat_timer.Q, pt:=t#10s);

FOR i:=0 TO (SIZEOF(data2floor)-1)-1 DO
	IF data2floor[i]<>data2floor_prev[i] THEN
		b_write2:=TRUE;
		EXIT;
	ELSE
		b_write2:=FALSE;
	END_IF
END_FOR

IF try_again2 AND NOT timer2.Q THEN
	b_write2:=TRUE;
	try_again2:=FALSE;
END_IF


IF write_ads2.BUSY THEN b_write2:=FALSE; END_IF

	write_ads2(
		NETID:=ads_adr2,
		PORT:=800,
		IDXGRP:=16#4020,
		IDXOFFS:=100,
		WRITE:=b_write2,
		TMOUT:=write_timeout,
		LEN:=SIZEOF(data2floor),
		SRCADDR:=ADR(data2floor));

IF write_ads2.ERR AND NOT timer2.Q THEN
	timer2.IN:=TRUE;
	try_again2:=TRUE;
END_IF
timer2(PT:=write_timeout);
timer2.IN:=FALSE;

FOR j:=0 TO (SIZEOF(data2floor)-1)-1 DO
	data2floor_prev[j]:=data2floor[j];
END_FOR

SENT2(CLK:=write_ads2.BUSY);

IF NOT write_ads2.ERR THEN
	SNT_CNT2(CU:=SENT2.Q);
END_IF

(*3floor*)
FOR i1:=0 TO (SIZEOF(data3floor)-1)-1DO
	IF data3floor[i1]<>data3floor_prev[i1] OR fb_heartbeat_timer.Q  THEN
		b_write3:=TRUE;
		EXIT;
	ELSE
		b_write3:=FALSE;
	END_IF
END_FOR

IF try_again3 AND NOT timer3.Q THEN
	b_write3:=TRUE;
	try_again3:=FALSE;
END_IF


IF write_ads3.BUSY THEN b_write3:=FALSE; END_IF

	write_ads3(
		NETID:=ads_adr3,
		PORT:=801,
		IDXGRP:=16#4020,
		IDXOFFS:=100,
		WRITE:=b_write3,
		TMOUT:=write_timeout,
		LEN:=SIZEOF(data3floor),
		SRCADDR:=ADR(data3floor));

IF write_ads3.ERR AND NOT timer3.Q THEN
	timer3.IN:=TRUE;
	try_again3:=TRUE;
END_IF
timer3(PT:=write_timeout);
timer3.IN:=FALSE;

SENT3(CLK:=write_ads3.BUSY);

IF NOT write_ads3.ERR THEN
	SNT_CNT3(CU:=SENT3.Q);
END_IF

FOR j1:=0 TO (SIZEOF(data3floor)-1)-1 DO
	data3floor_prev[j1]:=data3floor[j1];
END_FOR
END_PROGRAM
